(*********************************** G.D S.p.A. - Technical Department ***********************************
============= PROGRAM INFO ============
FOLDER:             TBD
MACHINES INVOLVED:  TBD 

============= DESCRIPTION =============
csp main interface program

============= REVISIONS ===============
Date		Version	 	Author      	Description             
----------	-------		------------  	--------------------------------------------
2019/09/27 	0000.00	 	M.Grasso		Creation of the PRG

**********************************************************************************************************)
PROGRAM _csp_case_glue_lowest
VAR
END_VAR

;

END_PROGRAM

(* stored: Version 1.1.0.1, ProductVersion 3.1.4022.12
   POU _csp_case_glue_lowest: Id {e656edf6-18ef-4ef2-a6e6-114332a75c8d}, SpecialFunc None *)
